FUNCTION_BLOCK PUBLISH_10 (* Publish to one or many SUBSCRIBE_10 Blocks *)
  (* Standard: 61499-2; Description: Copyright (c) 2017 fortiss GmbH This program and the accompanying materials are made available under the terms of the Eclipse Public License 2.0 which is available at https://www.eclipse.org/legal/epl-2.0/ SPDX-License-Identifier: EPL-2.0 *)
  (* Version 3.0, 2025-04-14, Patrick Aigner, changed package *)
  (* Version 1.0, 2017-10-25, Alois Zoitl, fortiss GmbH, initial API and implementation and/or initial documentation *)
  PACKAGE iec61499::net;
  {SET_ATTRIBUTE(eclipse4diac::core::GenericClassName, 'GEN_PUBLISH')}
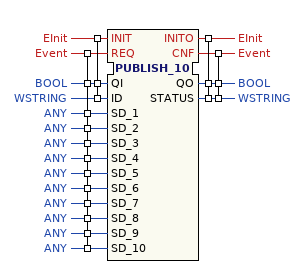
  EVENT_INPUT
    INIT : EInit WITH QI, ID; (* Initialization *)
    REQ WITH QI, SD_1, SD_2, SD_3, SD_4, SD_5, SD_7, SD_6, SD_8, SD_9, SD_10; (* Send Data, unconfirmed *)
  END_EVENT
  EVENT_OUTPUT
    INITO : EInit WITH QO, STATUS; (* Initialization Confirm *)
    CNF WITH QO, STATUS; (* Data was sent *)
  END_EVENT
  VAR_INPUT
    QI : BOOL;
    ID : WSTRING;
    SD_1 : ANY;
    SD_2 : ANY;
    SD_3 : ANY;
    SD_4 : ANY;
    SD_5 : ANY;
    SD_6 : ANY;
    SD_7 : ANY;
    SD_8 : ANY;
    SD_9 : ANY;
    SD_10 : ANY;
  END_VAR
  VAR_OUTPUT
    QO : BOOL;
    STATUS : WSTRING;
  END_VAR
END_FUNCTION_BLOCK
